// SIMATIC STEP 7 (V5.x) project DATE_TIME_READ
// CPU: CPU 319F-3 PN/DP
// station: Hardware
// station: SIMATIC 300
// station: P_ADR_BUS
// program: S7 Program(2)

SYMBOL_TABLE
"DATE_TIME_READ"	DB 1	DB 1	// DATE_TIME_READ
"DATE_TIME"	FC 1	FC 1	// DATE_TIME
"DAY_OF_WEEK"	FC 2	FC 2	// DAY_OF_WEEK
"DT_DATE"	FC 6	FC 6	// DT to DATE
"DT_DAY"	FC 7	FC 7	// DT to DAY
"DT_TOD"	FC 8	FC 8	// DT to TOD
"M10.0"	M 10.0	BOOL	// BIT MEMORY
"MW2"	MW 2	INT	// DIA_SEMANA
"MW21"	MW 21	INT	// MINUTO
"MW22"	MW 22	INT	// HORA
"Main Program"	OB 1	OB 1
"I/O_FLT1"	OB 82	OB 82	// I/O Point Fault 1
"RACK_FLT"	OB 86	OB 86	// Loss of Rack Fault
"PROG_ERR"	OB 121	OB 121	// Programming Error
"READ_CLK"	SFC 1	SFC 1	// Read System Clock
"RD_SINFO"	SFC 6	SFC 6	// Read OB Start Information
"VAT_1"	VAT 1	
END_SYMBOL_TABLE

FUNCTION "DATE_TIME" : VOID	// FC 1
AUTHOR : Cesar
VERSION : 0.1
BEGIN
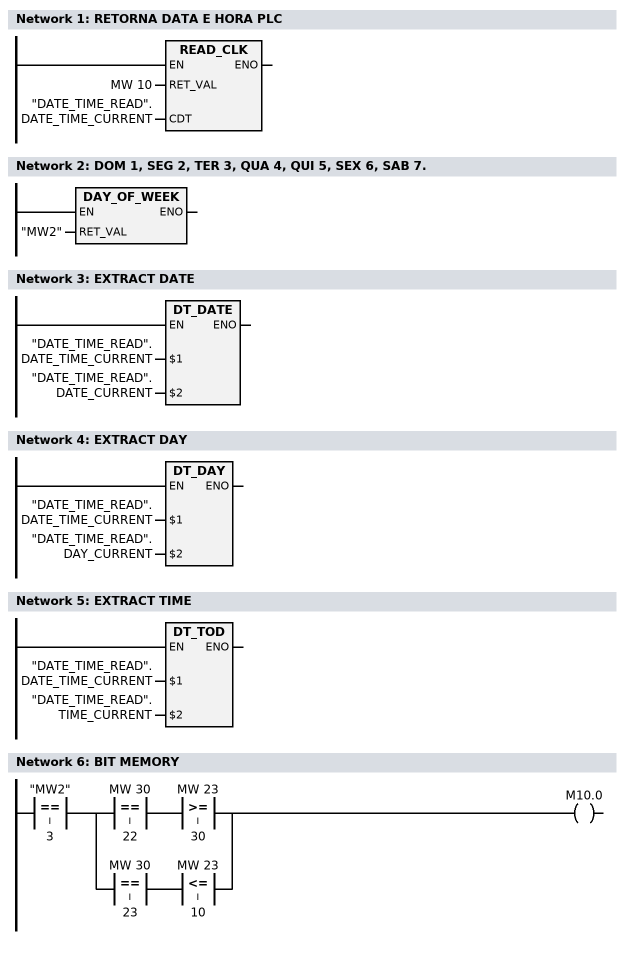
NETWORK
TITLE = RETORNA DATA E HORA PLC
      CALL  "READ_CLK" (
           RET_VAL                  := MW 10,
           CDT                      := "DATE_TIME_READ".DATE_TIME_CURRENT);
      NOP   0;
NETWORK
TITLE = DOM 1, SEG 2, TER 3, QUA 4, QUI 5, SEX 6, SAB 7.
      CALL  "DAY_OF_WEEK" (
           RET_VAL                  := "MW2");
      NOP   0;
NETWORK
TITLE = EXTRACT DATE
      CALL  "DT_DATE" (
           $1                       := "DATE_TIME_READ".DATE_TIME_CURRENT,
           $2                       := "DATE_TIME_READ".DATE_CURRENT);
      NOP   0;
NETWORK
TITLE = EXTRACT DAY
      CALL  "DT_DAY" (
           $1                       := "DATE_TIME_READ".DATE_TIME_CURRENT,
           $2                       := "DATE_TIME_READ".DAY_CURRENT);
      NOP   0;
NETWORK
TITLE = EXTRACT TIME
      CALL  "DT_TOD" (
           $1                       := "DATE_TIME_READ".DATE_TIME_CURRENT,
           $2                       := "DATE_TIME_READ".TIME_CURRENT);
      NOP   0;
NETWORK
TITLE = BIT MEMORY
      A(;
      L     "MW2";
      L     3;
      ==I;
      );
      A(;
      A(;
      L     MW 30;
      L     22;
      ==I;
      );
      A(;
      L     MW 23;
      L     30;
      >=I;
      );
      O;
      A(;
      L     MW 30;
      L     23;
      ==I;
      );
      A(;
      L     MW 23;
      L     10;
      <=I;
      );
      );
      =     "M10.0";
END_FUNCTION

FUNCTION "DAY_OF_WEEK" : INT	// FC 2
TITLE = DAY OF WEEK
//(C)Copyright Cesar Netto 2025 - 2025
//--------------------------------------------------------------------------------
//Title:              FC_DayOfWeek
//Comment/Function:   Retorna o dia da semana com base em dados da CPU (RTC), 
//incluindo conversão de BCD para inteiro.
//Library/Family:     Utilitários de Data e Hora
//Author:             Cesar Netto / Engenharia de Automação
//Tested on System:   S7-300/400 CPU 319F-3 PN/DP FW 2.8 (Testado em PLCSIM e 
//ambiente real)
//Engineering:        Simatic Manager V5.6 SP1
//Restrictions:       Utilizar em OB1 ou blocos chamados por OB1. Não compatível 
//com S7-1200 sem ajustes de RTC.
//Requirements:       Controlador com acesso à área de tempo real (RTC). Nenhum 
//pacote adicional necessário.
//
//--------------------------------------------------------------------------------
//Change log table:
//Version     | Date       | Signature   | Expert in charge   | Changes applied
//------------|------------|-------------|--------------------|----------------
//001.000.000 | 2025-08-05 | ----------  | Cesar Netto        | First release
AUTHOR : CESAR
VERSION : 0.1
VAR_OUTPUT
  RET_VAL : INT ;
END_VAR
VAR_TEMP
  YY : INT ;
  MM : INT ;
  DD : INT ;
  AR1 : INT ;
  AR2 : INT ;
  AR3 : INT ;
  AR4 : INT ;
  AR5 : INT ;
  AR6 : INT ;
END_VAR
BEGIN
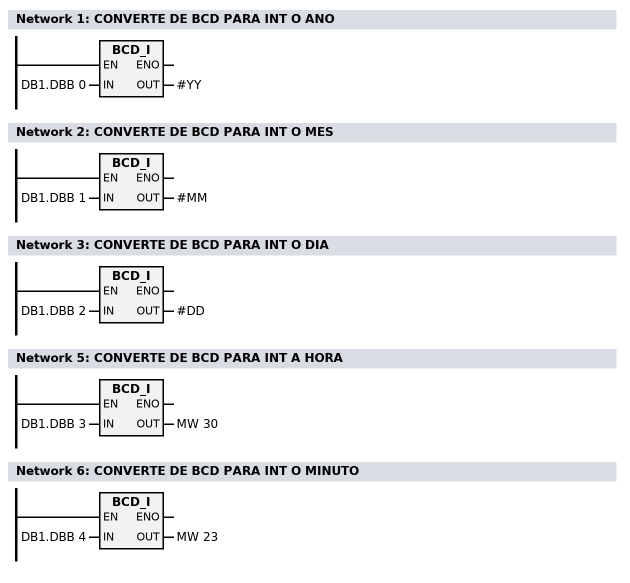
NETWORK
TITLE = CONVERTE DE BCD PARA INT O ANO
      L     DB1.DBB 0;
      BTI;
      T     #YY;
NETWORK
TITLE = CONVERTE DE BCD PARA INT O MES
      L     DB1.DBB 1;
      BTI;
      T     #MM;
NETWORK
TITLE = CONVERTE DE BCD PARA INT O DIA
      L     DB1.DBB 2;
      BTI;
      T     #DD;
NETWORK
TITLE = CALCULO DIA DA SEMANA
// (network holds code this reader does not know; not shown)
// SOMA
NETWORK
TITLE = CONVERTE DE BCD PARA INT A HORA
      L     DB1.DBB 3;
      BTI;
      T     MW 30;
      NOP   0;
NETWORK
TITLE = CONVERTE DE BCD PARA INT O MINUTO
      L     DB1.DBB 4;
      BTI;
      T     MW 23;
      NOP   0;
END_FUNCTION

// FC 6: know-how protected block, not included

// FC 7: know-how protected block, not included

// FC 8: know-how protected block, not included

DATA_BLOCK "DATE_TIME_READ"	// DB 1
AUTHOR : Cesar
VERSION : 0.1
  STRUCT
   DATE_TIME_CURRENT : DATE_AND_TIME ;
   DATE_CURRENT : DATE ;
   DAY_CURRENT : INT ;
   TIME_CURRENT : TIME_OF_DAY ;
  END_STRUCT ;	
BEGIN
END_DATA_BLOCK

ORGANIZATION_BLOCK "Main Program"	// OB 1
TITLE = "Main Program Sweep (Cycle)"
AUTHOR : Cesar
VERSION : 0.1
VAR_TEMP
  OB1_EV_CLASS : BYTE ;	//Bits 0-3 = 1 (Coming event), Bits 4-7 = 1 (Event class 1)
  OB1_SCAN_1 : BYTE ;	//1 (Cold restart scan 1 of OB 1), 3 (Scan 2-n of OB 1)
  OB1_PRIORITY : BYTE ;	//Priority of OB Execution
  OB1_OB_NUMBR : BYTE ;	//1 (Organization block 1, OB1)
  OB1_RESERVED_1 : BYTE ;	//Reserved for system
  OB1_RESERVED_2 : BYTE ;	//Reserved for system
  OB1_PREV_CYCLE : INT ;	//Cycle time of previous OB1 scan (milliseconds)
  OB1_MIN_CYCLE : INT ;	//Minimum cycle time of OB1 (milliseconds)
  OB1_MAX_CYCLE : INT ;	//Maximum cycle time of OB1 (milliseconds)
  OB1_DATE_TIME : DATE_AND_TIME ;	//Date and time OB1 started
END_VAR
BEGIN
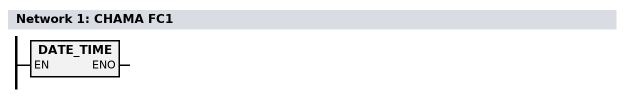
NETWORK
TITLE = CHAMA FC1
      CALL  "DATE_TIME";
      NOP   0;
END_ORGANIZATION_BLOCK

ORGANIZATION_BLOCK "I/O_FLT1"	// OB 82
TITLE = "I/O Point Fault"
VERSION : 0.1
VAR_TEMP
  OB82_EV_CLASS : BYTE ;	//16#39, Event class 3, Entering event state, Internal fault event
  OB82_FLT_ID : BYTE ;	//16#XX, Fault identifcation code
  OB82_PRIORITY : BYTE ;	//Priority of OB Execution
  OB82_OB_NUMBR : BYTE ;	//82 (Organization block 82, OB82)
  OB82_RESERVED_1 : BYTE ;	//Reserved for system
  OB82_IO_FLAG : BYTE ;	//Input (01010100), Output (01010101)
  OB82_MDL_ADDR : WORD ;	//Base address of module with fault
  OB82_MDL_DEFECT : BOOL ;	//Module defective
  OB82_INT_FAULT : BOOL ;	//Internal fault
  OB82_EXT_FAULT : BOOL ;	//External fault
  OB82_PNT_INFO : BOOL ;	//Point information
  OB82_EXT_VOLTAGE : BOOL ;	//External voltage low
  OB82_FLD_CONNCTR : BOOL ;	//Field wiring connector missing
  OB82_NO_CONFIG : BOOL ;	//Module has no configuration data
  OB82_CONFIG_ERR : BOOL ;	//Module has configuration error
  OB82_MDL_TYPE : BYTE ;	//Type of module
  OB82_SUB_MDL_ERR : BOOL ;	//Sub-Module is missing or has error
  OB82_COMM_FAULT : BOOL ;	//Communication fault
  OB82_MDL_STOP : BOOL ;	//Module is stopped
  OB82_WTCH_DOG_FLT : BOOL ;	//Watch dog timer stopped module
  OB82_INT_PS_FLT : BOOL ;	//Internal power supply fault
  OB82_PRIM_BATT_FLT : BOOL ;	//Primary battery is in fault
  OB82_BCKUP_BATT_FLT : BOOL ;	//Backup battery is in fault
  OB82_RESERVED_2 : BOOL ;	//Reserved for system
  OB82_RACK_FLT : BOOL ;	//Rack fault, only for bus interface module
  OB82_PROC_FLT : BOOL ;	//Processor fault
  OB82_EPROM_FLT : BOOL ;	//EPROM fault
  OB82_RAM_FLT : BOOL ;	//RAM fault
  OB82_ADU_FLT : BOOL ;	//ADU fault
  OB82_FUSE_FLT : BOOL ;	//Fuse fault
  OB82_HW_INTR_FLT : BOOL ;	//Hardware interupt input in fault
  OB82_RESERVED_3 : BOOL ;	//Reserved for system
  OB82_DATE_TIME : DATE_AND_TIME ;	//Date and time OB82 started
END_VAR
BEGIN
// (block stored without names or comments; labels and parameter names are numbered)
END_ORGANIZATION_BLOCK

ORGANIZATION_BLOCK "RACK_FLT"	// OB 86
TITLE = "Loss Of Rack Fault"
VERSION : 0.1
VAR_TEMP
  OB86_EV_CLASS : BYTE ;	//16#38/39 Event class 3
  OB86_FLT_ID : BYTE ;	//16#C1/C4/C5, Fault identifcation code
  OB86_PRIORITY : BYTE ;	//Priority of OB Execution
  OB86_OB_NUMBR : BYTE ;	//86 (Organization block 86, OB86)
  OB86_RESERVED_1 : BYTE ;	//Reserved for system
  OB86_RESERVED_2 : BYTE ;	//Reserved for system
  OB86_MDL_ADDR : WORD ;	//Base address of IM module in rack with fault
  OB86_RACKS_FLTD : ARRAY  [0 .. 31 ] OF BOOL ;	//Racks in fault
  OB86_DATE_TIME : DATE_AND_TIME ;	//Date and time OB86 started
END_VAR
BEGIN
// (block stored without names or comments; labels and parameter names are numbered)
END_ORGANIZATION_BLOCK

ORGANIZATION_BLOCK "PROG_ERR"	// OB 121
TITLE = "Programming Error"
VERSION : 0.1
VAR_TEMP
  OB121_EV_CLASS : BYTE ;	//16#25, Event class 2, Entering event state, Internal fault event
  OB121_SW_FLT : BYTE ;	//16#XX Software programming fault
  OB121_PRIORITY : BYTE ;	//Priority of OB Execution
  OB121_OB_NUMBR : BYTE ;	//121 (Organization block 121, OB121)
  OB121_BLK_TYPE : BYTE ;	//16#88/8A/8B/8C/8E Type of block fault occured in
  OB121_RESERVED_1 : BYTE ;	//Reserved for system
  OB121_FLT_REG : WORD ;	//16#XX Specific register that caused fault
  OB121_BLK_NUM : WORD ;	//Number of block that programming fault occured in
  OB121_PRG_ADDR : WORD ;	//Address in block where programming fault occured
  OB121_DATE_TIME : DATE_AND_TIME ;	//Date and time OB121 started
END_VAR
BEGIN
// (block stored without names or comments; labels and parameter names are numbered)
END_ORGANIZATION_BLOCK
